TYPE
    ST_MyComponent_HMI : STRUCT
        Config  : ST_MyComponent_Config;
        Command : ST_MyComponent_Command;
        Status  : ST_MyComponent_Status;
    END_STRUCT
END_TYPE

(* stored: Version 1.1.0.1
   DUT ST_MyComponent_HMI: Id {b67c2710-1a47-4261-aeef-e6b49bbcd616} *)
